FUNCTION F_ParsePayload : STRING(160)
VAR_INPUT 
	rx:STRING(255); 
END_VAR
VAR 
	i:INT; 
	sData:STRING(160); 
	p1,p2:INT; 
END_VAR

p1:=0; 
p2:=0;

FOR i:=1 TO LEN(rx) DO
	IF TO_BYTE(rx[i])=GVL_CONSTANT.cSTX THEN 
		p1:=i; 
	END_IF
	
	IF TO_BYTE(rx[i])=GVL_CONSTANT.cETX THEN 
		p2:=i; 
		EXIT; 
	END_IF
END_FOR
IF (p1>0) AND (p2>p1) THEN 
	sData := MID(rx, p1+1, p2-(p1+1)); 
END_IF
F_ParsePayload := sData;

END_FUNCTION

(* stored: Version 1.1.0.1, ProductVersion 3.1.4024.15
   POU F_ParsePayload: Id {f5d1633d-d515-49d3-a0d8-fa9724045037}, SpecialFunc None *)
